(* IEC 61131-3 sources: UERANSIM_with_OpenPLC/, 2 files *)

(* ---- 1st_basic.st ---- *)
PROGRAM program0
  VAR
    SWITCH AT %QX0.0 : BOOL;
    SLAVE1 AT %QW0 : INT;
  END_VAR
  VAR
    setpoint : INT := 10;
    GT2_OUT : BOOL;
  END_VAR

  GT2_OUT := GT(SLAVE1, setpoint);
  SWITCH := GT2_OUT;
END_PROGRAM

CONFIGURATION Config0

  RESOURCE Res0 ON PLC
    TASK task0(INTERVAL := T#20ms,PRIORITY := 0);
    PROGRAM instance0 WITH task0 : program0;
  END_RESOURCE
END_CONFIGURATION

(* ---- 2nd_complex.st ---- *)
PROGRAM program0
  VAR
    SWITCH AT %QX0.0 : BOOL;
  END_VAR
  VAR
    setpoint : INT := 10;
    GT2_OUT : BOOL;
  END_VAR
  VAR
    SLAVE1 AT %QW150 : INT := 11;
    PARVO AT %QW151 : INT;
  END_VAR

  GT2_OUT := GT(SLAVE1, setpoint);
  SWITCH := GT2_OUT;
  IF SWITCH=TRUE THEN
    PARVO := 1;
  ELSE
    PARVO := 0;
  END_IF;

END_PROGRAM

CONFIGURATION Config0

  RESOURCE Res0 ON PLC
    TASK task0(INTERVAL := T#20ms,PRIORITY := 0);
    PROGRAM instance0 WITH task0 : program0;
  END_RESOURCE
END_CONFIGURATION
